(* CODESYS project WashingMachineVisu.export

Project tree, tasks and I/O mapping:
  visualisation Visualization
*)

// /Visualization
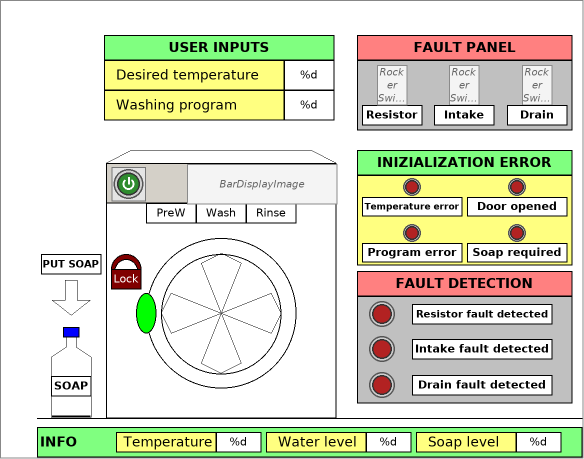
VISUALIZATION Visualization  // 584x459
    Line (37,418) (582,418)
    Rectangle (106,178 230x240)
    Ellipse (162,254 118x118)
    Rectangle (161,255 120x120)
        p1126004900: -GVL.waterlevel/3*2
    Ellipse (146,238 150x150)
    Ellipse (161,254 120x120)
    Polygon (221,253) (201,263) (221,313) (171,293) (161,313) (171,333) (221,313) (201,363) (221,373) (241,363) (221,313) (271,333) (281,313) (271,293) (221,313) (241,263)
        p2858320360: GVL.motor
    Ellipse (136,293 20x40), colour toggle: GVL.bulls_eye_open
        toggle GVL.bulls_eye_open
    Ellipse (111,254 30x30), colour toggle: GVL.bulls_eye_lock
    Ellipse (114,259 24x27)
    Rectangle (111,269 30x20), "Lock", colour toggle: GVL.bulls_eye_lock
    Rectangle (106,163 230x40)
    Rectangle (146,203 50x20), "PreW", colour toggle: GVL.prewash
    Rectangle (196,203 50x20), "Wash", colour toggle: GVL.wash
    Rectangle (246,203 50x20), "Rinse", colour toggle: GVL.rinse
    Polygon (106,163) (131,150) (311,150) (336,163)
    PowerSwitch (111,167 35x34), variable: GVL.run, behaviour: TOGGLE, style: Switch-PowerSwitch-Green
    BarDisplayImage (187,164 150x40), value: GVL.temperature, style: BarDisplayImage-Gray, scale format: %.0f, scale 0..90
    Polygon (51,417) (51,357) (66,347) (66,332) (76,332) (76,347) (91,357) (91,417)
    Rectangle (63,327 16x10)
    Rectangle (104,60 180x30), "Desired temperature"
        OnMouseDown: write GVL.temp_number via VisuDialogs.Numpad, min 0, max 100, format 0
    Rectangle (104,90 180x30), "Washing program"
        OnMouseDown: write GVL.prog_number via VisuDialogs.Numpad, min 0, max 100, format 0
    Rectangle (104,35 230x25), "USER INPUTS"
    Rectangle (284,60 50x30), "%d", text variable: GVL.temp_number
    Rectangle (284,90 50x30), "%d", text variable: GVL.prog_number
    Rectangle (37,427 545x30), "INFO"
    Rectangle (116,432 100x20), "Temperature"
    Rectangle (357,150 215x25), "INIZIALIZATION ERROR"
    Rectangle (216,432 45x20), "%d", text variable: GVL.temperature
    Rectangle (266,432 100x20), "Water level"
    Rectangle (366,432 45x20), "%d", text variable: GVL.waterlevel
    Rectangle (416,432 100x20), "Soap level"
    Rectangle (516,432 45x20), "%d", text variable: GVL.soaplevel
    Rectangle (357,175 215x90)
    Lamp1 (402,177 20x20), variable: GVL.temp_error, style: Lamp-Lamp1-Red
    Rectangle (362,197 100x19), "Temperature error"
    Lamp1 (507,177 20x20), variable: GVL.bulls_eye_open, style: Lamp-Lamp1-Red
    Rectangle (467,197 100x19), "Door opened"
    Lamp1 (402,223 20x20), variable: GVL.prog_error, style: Lamp-Lamp1-Red
    Rectangle (362,243 100x19), "Program error"
    Lamp1 (507,223 20x20), variable: GVL.soap_alarm, style: Lamp-Lamp1-Red
    Rectangle (467,243 100x19), "Soap required"
    Rectangle (357,35 215x25), "FAULT PANEL"
    Rectangle (357,60 215x70)
    Rectangle (362,105 60x20), "Resistor"
    RockerSwitch (377,65 30x40), variable: GVL.heat_fail, behaviour: TOGGLE, style: Switch-RockerSwitch-Red
    RockerSwitch (449,65 30x40), variable: GVL.water_in_fail, behaviour: TOGGLE, style: Switch-RockerSwitch-Red
    Rectangle (434,105 60x20), "Intake"
    RockerSwitch (522,65 30x40), variable: GVL.water_out_fail, behaviour: TOGGLE, style: Switch-RockerSwitch-Red
    Rectangle (507,105 60x20), "Drain"
    Rectangle (357,271 215x25), "FAULT DETECTION"
    Rectangle (357,296 215x107)
    Lamp1 (367,299 30x30), variable: GVL.heat_alarm, style: Lamp-Lamp1-Red
    Rectangle (412,304 140x20), "Resistor fault detected"
    Lamp1 (367,370 30x30), variable: GVL.water_out_alarm, style: Lamp-Lamp1-Red
    Lamp1 (367,334 30x30), variable: GVL.water_in_alarm, style: Lamp-Lamp1-Red
    Rectangle (412,339 140x20), "Intake fault detected"
    Rectangle (412,375 140x20), "Drain fault detected"
    Rectangle (52,416 38x0)
        p2773130477: -GVL.soaplevel
    Rectangle (51,376 40x20), "SOAP"
    Polygon (65,280) (65,300) (52,300) (71,315) (90,300) (77,300) (77,280), colour toggle: GVL.fillsoap
        toggle GVL.fillsoap
    Rectangle (41,254 60x20), "PUT SOAP"
END_VISUALIZATION
